DATA_BLOCK "PalletRelease"
{ S7_Optimized_Access := 'FALSE' }
VERSION : 0.1
NON_RETAIN
   STRUCT
      Buffer : Struct
         AskPallet : Bool;
         UnloadFlag : Bool;
      END_STRUCT;
      LaserMarking : Struct
         AskPallet : Bool;
         UnloadFlag : Bool;
      END_STRUCT;
      Print : Struct
         AskPallet : Bool;
         UnloadFlag : Bool;
      END_STRUCT;
      Spare : Struct
         AskPallet : Bool;
         UnloadFlag : Bool;
      END_STRUCT;
      Spare2 : Struct
         AskPallet : Bool;
         UnloadFlag : Bool;
      END_STRUCT;
      "Time" {InstructionName := 'TOF_TIME'; LibVersion := '1.0'; S7_SetPoint := 'False'} : Array[0..1] of TOF_TIME;
      LaserMarkingBuffer { S7_SetPoint := 'False'} : "LaserMarkingBuffer";
   END_STRUCT;


BEGIN

END_DATA_BLOCK

